{attribute 'Tc2GvlVarNames'}
VAR_GLOBAL CONSTANT
	(* analog_actuator define *)
	ANALOG_ACTUATOR_CLASS_NAME:		STRING := 'analog_actuator';
	ANALOG_ACTUATOR_MAX_TEST_COMMANDS:	DINT :=	2;
END_VAR

VAR_GLOBAL
END_VAR

(* stored: Version 1.1.0.1, ProductVersion 3.1.4022.12
   GVL analog_actuator_global: Id {a7dfa2ea-06d4-4a67-9dc2-85db4483c4e2} *)
